(* PLC project Generated.project, CODESYS CODESYS V3.5 SP19 Patch 1 *)
(* stored: creationDateTime 2026-09-06T13:00:42.480247, modificationDateTime 2026-09-06T13:00:42.480247 *)

TYPE ST_ChainBucket : STRUCT
  Idx101_BucketIsOpen : BOOL;  (* 1 = Benne Mécaniquement Ouvert | 0 = Non Confirmé *)
  Idx102_BucketIsClosed : BOOL;  (* 1 = Benne Mécaniquement Fermé | 0 = Non Confirmé *)
  Idx103_OffsetPos_M : REAL;  (* [mètres] Écart d'Ouverture Câble M1/M2 *)
  Idx104_AutoSeqActive : BOOL;  (* : 1 = Séquencement auto (ouverture/fermeture armée par mouvement couplé) en cours *)
  Idx105_StateIncoherent : BOOL;  (* : 1 = État ouvert/fermé INCONNU (ni IsOpen ni IsClosed fiable) -- cause fréquente de blocage *)
  Idx106_FBState : E_State;  (* : État machine FB_Bucket (READY/BUSY/DONE/DISABLED) *)
  Idx107_LastPosM2Open_M : REAL;  (* : Dernière position M2 mémorisée "ouvert" *)
  Idx108_LastPosM2Close_M : REAL;  (* : Dernière position M2 mémorisée "fermé" *)
  Idx109_BucketTooOpen : BOOL;  (* ⚠️ Dépassement ouverture : Delta < OffsetOpen - Tolerance (Enrouler M2) *)
  Idx110_BucketTooClosed : BOOL;  (* ⚠️ Dépassement fermeture : Delta > OffsetClose + Tolerance (Dérouler M2) *)
  Idx111_BucketIsIntermediate : BOOL;  (* ↔️ Position intermédiaire (entrebâillée entre ouvert et fermé) *)
  Idx112_DeltaPosition_M : REAL;  (* 📏 Écart réel signé M2 - M1 (mètres) en direct *)
  Idx113_MachineHomed : BOOL;  (* Reference M1/M2/benne qualifiee *)
  Idx114_MachineHomingStep : INT;  (* Etape guidee reference machine *)
  Idx115_MachineHomingFailed : BOOL;  (* Transaction reference abandonnee *)
  Idx116_M1ReferenceMissing : BOOL;  (* M1 non reference ou mesure douteuse *)
  Idx117_M2ReferenceMissing : BOOL;  (* M2 non reference ou mesure douteuse *)
  Idx118_BucketOffsetUnknown : BOOL;  (* Offset benne non confirme *)
  Idx119_ReferenceTransaction : BOOL;  (* Homing conjoint en cours *)
  Idx120_MachineHomingLossSafeStop : BOOL;  (* Perte reference pendant mouvement *)
  Idx201_HmiCmd_BtnOpen : BOOL;  (* 1 = Demande Ouverture IHM | 0 = Relâché *)
  Idx202_HmiCmd_BtnClose : BOOL;  (* 1 = Demande Fermeture IHM | 0 = Relâché *)
  Idx203_CycleCmd_Open : BOOL;  (* 1 = Demande Ouverture par le Cycle Auto *)
  Idx204_CoupledDiveOpenArmed : BOOL;  (* : 1 = Ouverture auto armée (descente couplée demandée, benne pas ouverte) *)
  Idx205_CoupledAscentCloseArmed : BOOL;  (* : 1 = Fermeture auto armée (montée couplée demandée, benne pas fermée) *)
  Idx206_CloseReqActive : BOOL;  (* : 1 = Fermeture mémorisée/en cours (instBucket.CloseReq -- reste à 1 si recul partiel non terminé) *)
  Idx207_OpenReqActive : BOOL;  (* : 1 = Ouverture mémorisée/en cours (instBucket.OpenReq -- idem) *)
  Idx208_MotionBlockedByBucket : BOOL;  (* : 1 = Mouvement couplé BLOQUÉ (auto-séquencement armé mais benne pas Busy -- vérifier Idx306_ErrorIdRaw) *)
  Idx301_EmergencyChainClosed : BOOL;  (* 1 = Boucle Urgence OK | 0 = AU Appuyé *)
  Idx302_BucketFaultActive : BOOL;  (* 0 = Sain | 1 = Défaut Mouvement Benne *)
  Idx303_KoboldAutoStopEnabled : BOOL;  (* 1 = Toggle IHM arrêt auto descente actif *)
  Idx304_KoboldImmersionConfirmed : BOOL;  (* : 1 = Immersion confirmée (front Kobold dans la fenêtre) *)
  Idx305_KoboldBottomTouchLatched : BOOL;  (* : 1 = Fond détecté, descente bloquée (ProcessPermitM1/M2_Descend) *)
  Idx306_ErrorIdRaw : WORD;  (* : bitfield brut FB_Bucket (bit0 configuration, bit1 écart M2/M1, bit2 timeout, bit3 glissement M1, bit4 codeurs non référencés) *)
  Idx307_EffectivePermit_Open : BOOL;  (* 1 = ouverture benne physiquement autorisée *)
  Idx308_EffectivePermit_Close : BOOL;  (* 1 = fermeture benne physiquement autorisée *)
  Idx401_BucketBusy : BOOL;  (* 1 = Mouvement Mâchoires en cours | 0 = Repos *)
  Idx402_BucketDone : BOOL;  (* 1 = Position Cible Atteinte | 0 = En cours *)
  Idx403_ExtractionControlActive : BOOL;  (* : 1 = Phase vitesse contrôlée montée en cours *)
  Idx501_M2_CmdRev_DQ : BOOL;  (* 1 = Relais Action Benne M2 ON *)
END_STRUCT;
END_TYPE

(* values of E_State: DISABLED: Enable faux, neutralisé; INIT: Démarrage / vérifs; READY: Prêt, attend ordre; BUSY: Action en cours; DONE: Action terminée; STOPPING: Décél rampe avant arrêt (StartStop=FALSE ou SafeStop=TRUE); ERROR: Défaut actif non acquitté (FB en erreur — HMI non aveugle) *)

{attribute 'qualified_only'}
{attribute 'strict'}
TYPE E_State : (DISABLED := 0, INIT := 1, READY := 2, BUSY := 3, DONE := 4, STOPPING := 5, ERROR := 6);
END_TYPE
